// TIA Portal V20 export
// export: Created 2025-12-01T14:56:59.3447129Z, ExportSetting None, DisplayName Totally Integrated Automation Portal, DisplayVersion V20 Update 3, DisplayName TIA Portal Openness, DisplayVersion V20 Update 3, DisplayName TIA Portal Version Control Interface, DisplayVersion V20 Update 3, DisplayName STEP 7 Professional, DisplayVersion V20 Update 3, DisplayName STEP 7 Safety, DisplayVersion V20 Update 2, DisplayName WinCC Basic/Comfort/Advanced, DisplayVersion V20 Update 3, DisplayName WinCC Professional, DisplayVersion V20 Update 3, DisplayName WinCC Unified, DisplayVersion V20 Update 3
FUNCTION "FC402_Conector_ZONA_HB" : Void   // FC402, LAD
{ S7_Optimized_Access := 'FALSE' }
AUTHOR : TLigero
NAME : 20160208
VERSION : 3.1
// stored: AutoNumber false, SetENOAutomatically false
   VAR_INPUT
      Mesa : UInt;
      En_Tension : Bool;
      HB_B_INI : Bool;
      HB_Avance_INI : Bool;
      HB_B_FIN : Bool;
      HB_Avance_FIN : Bool;
      Zona_HB_OK : Bool;
      PRV_AVTF : Bool;
      NXT_Carga_OK : Bool;
      NXT_Avance : Bool;
      V_Paro_Tms : UDInt;
      V_Seg_HB_Avance_Tms : UDInt;
      V_CNTSeparacion : UDInt;
   END_VAR
   VAR_OUTPUT
      PRV_Carga_OK : Bool;
      NXT_AVTF : Bool;
   END_VAR
   VAR_IN_OUT
      Mem_CNT_Tmp_Paro_Tx : Bool;
      Mem_CNT_Seg_HB_Avance : Bool;
      Maux_FN : Bool;
      MemAuxFN_HBpHs : Bool;
   END_VAR
   VAR_TEMP
      OK_Separacion_salida : Bool;
      FN_HBpHs : Bool;
      OK_sep_entrada : Bool;
      TEMP_HB_PTF_Desc : Bool;
      Ok_Tension : Bool;
      EstadoVI : "EstadosMesa";   // Estado del Vehiculo Inteliguente de la Mesa
   END_VAR
   VAR_TEMP   // added for the SCL form of the ladder/FBD networks
      _w1 : Bool;
   END_VAR
BEGIN

REGION Network 1
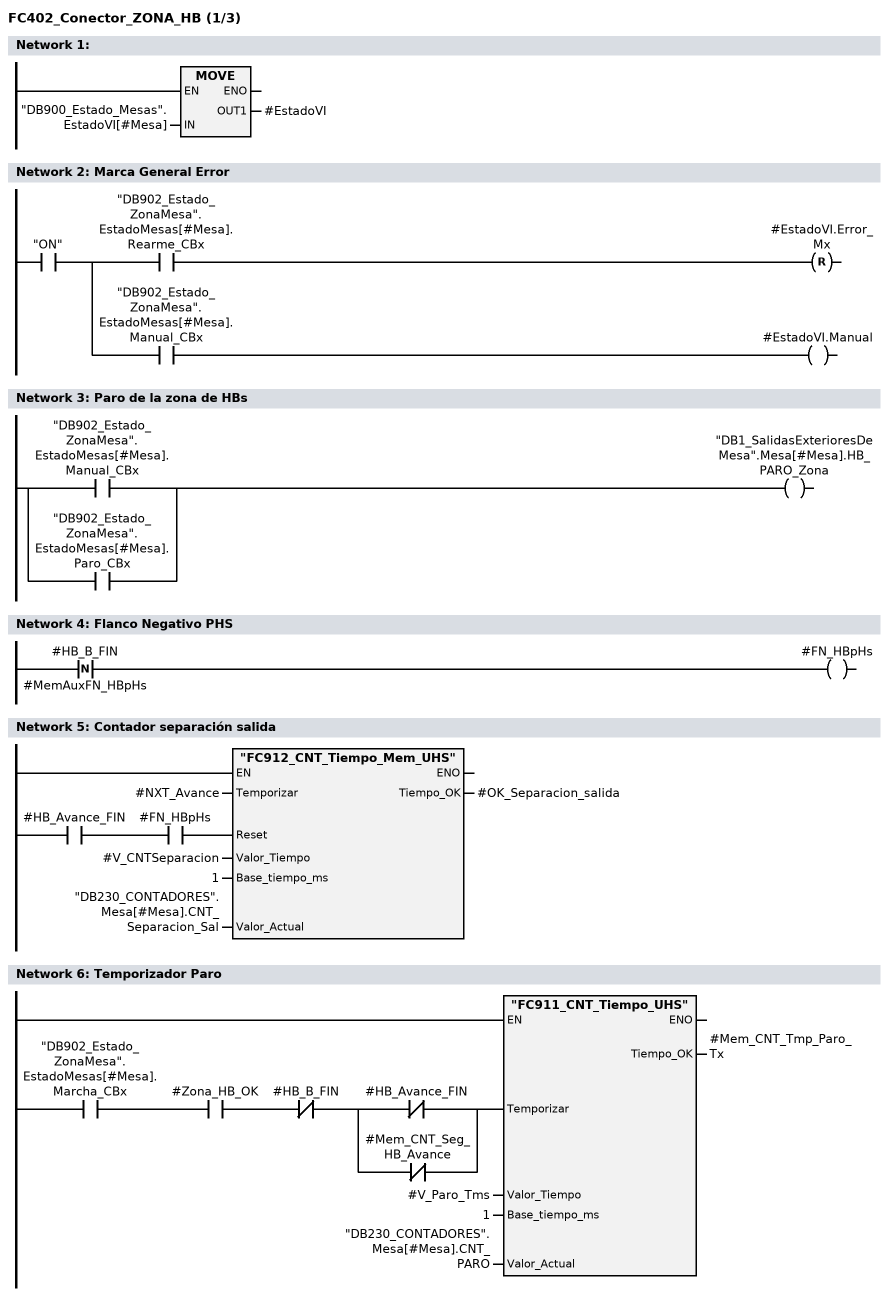
   RUNG wire#powerrail
      Move(in := "DB900_Estado_Mesas".EstadoVI[#Mesa], out1 => #EstadoVI)
   END_RUNG
   // the same network as SCL:
   #EstadoVI := "DB900_Estado_Mesas".EstadoVI[#Mesa];
END_REGION

REGION Network 2: Marca General Error
   RUNG wire#powerrail
      Contact( "ON" )
      wire#w1
      Contact( "DB902_Estado_ZonaMesa".EstadoMesas[#Mesa].Rearme_CBx )
      R_Coil( #EstadoVI.Error_Mx )
   END_RUNG
   RUNG wire#w1
      Contact( "DB902_Estado_ZonaMesa".EstadoMesas[#Mesa].Manual_CBx )
      Coil( #EstadoVI.Manual )
   END_RUNG
   // the same network as SCL:
   IF "ON" AND "DB902_Estado_ZonaMesa".EstadoMesas[#Mesa].Rearme_CBx THEN
       #EstadoVI.Error_Mx := FALSE;
   END_IF;
   #EstadoVI.Manual := "ON" AND "DB902_Estado_ZonaMesa".EstadoMesas[#Mesa].Manual_CBx;
END_REGION

REGION Network 3: Paro de la zona de HBs
   RUNG wire#powerrail
      Contact( "DB902_Estado_ZonaMesa".EstadoMesas[#Mesa].Manual_CBx )
      wire#w1
      Coil( "DB1_SalidasExterioresDeMesa".Mesa[#Mesa].HB_PARO_Zona )
   END_RUNG
   RUNG wire#powerrail
      Contact( "DB902_Estado_ZonaMesa".EstadoMesas[#Mesa].Paro_CBx )
   END_RUNG wire#w1
   // the same network as SCL:
   "DB1_SalidasExterioresDeMesa".Mesa[#Mesa].HB_PARO_Zona := "DB902_Estado_ZonaMesa".EstadoMesas[#Mesa].Manual_CBx OR "DB902_Estado_ZonaMesa".EstadoMesas[#Mesa].Paro_CBx;
END_REGION

REGION Network 4: Flanco Negativo PHS
   RUNG wire#powerrail
      N_Contact(operand := #HB_B_FIN, bit := #MemAuxFN_HBpHs)
      Coil( #FN_HBpHs )
   END_RUNG
   // the same network as SCL:
   #_w1 := NOT #HB_B_FIN AND #MemAuxFN_HBpHs;   // falling edge of #HB_B_FIN
   #MemAuxFN_HBpHs := #HB_B_FIN;
   #FN_HBpHs := #_w1;
END_REGION

REGION Network 5: Contador separación salida
   RUNG wire#powerrail
      "FC912_CNT_Tiempo_Mem_UHS"(Reset := wire#w1, Temporizar := #NXT_Avance, Valor_Tiempo := #V_CNTSeparacion, Base_tiempo_ms := 1, Valor_Actual := "DB230_CONTADORES".Mesa[#Mesa].CNT_Separacion_Sal, Tiempo_OK => #OK_Separacion_salida)
   END_RUNG
   RUNG wire#powerrail
      Contact( #HB_Avance_FIN )
      Contact( #FN_HBpHs )
   END_RUNG wire#w1
   // the same network as SCL:
   "FC912_CNT_Tiempo_Mem_UHS"(Temporizar := #NXT_Avance,
                           Reset := #HB_Avance_FIN AND #FN_HBpHs,
                           Valor_Tiempo := #V_CNTSeparacion,
                           Base_tiempo_ms := 1,
                           Valor_Actual := "DB230_CONTADORES".Mesa[#Mesa].CNT_Separacion_Sal,
                           Tiempo_OK => #OK_Separacion_salida);
END_REGION

REGION Network 6: Temporizador Paro
   RUNG wire#powerrail
      "FC911_CNT_Tiempo_UHS"(Temporizar := wire#w2, Valor_Tiempo := #V_Paro_Tms, Base_tiempo_ms := 1, Valor_Actual := "DB230_CONTADORES".Mesa[#Mesa].CNT_PARO, Tiempo_OK => #Mem_CNT_Tmp_Paro_Tx)
   END_RUNG
   RUNG wire#powerrail
      Contact( "DB902_Estado_ZonaMesa".EstadoMesas[#Mesa].Marcha_CBx )
      Contact( #Zona_HB_OK )
      I_Contact( #HB_B_FIN )
      wire#w1
      I_Contact( #HB_Avance_FIN )
   END_RUNG wire#w2
   RUNG wire#w1
      I_Contact( #Mem_CNT_Seg_HB_Avance )
   END_RUNG wire#w2
   // the same network as SCL:
   "FC911_CNT_Tiempo_UHS"(Temporizar := "DB902_Estado_ZonaMesa".EstadoMesas[#Mesa].Marcha_CBx AND #Zona_HB_OK AND NOT #HB_B_FIN AND (NOT #HB_Avance_FIN OR NOT #Mem_CNT_Seg_HB_Avance),
                          Valor_Tiempo := #V_Paro_Tms,
                          Base_tiempo_ms := 1,
                          Valor_Actual := "DB230_CONTADORES".Mesa[#Mesa].CNT_PARO,
                          Tiempo_OK => #Mem_CNT_Tmp_Paro_Tx);
END_REGION

REGION Network 7: Permiso descarga
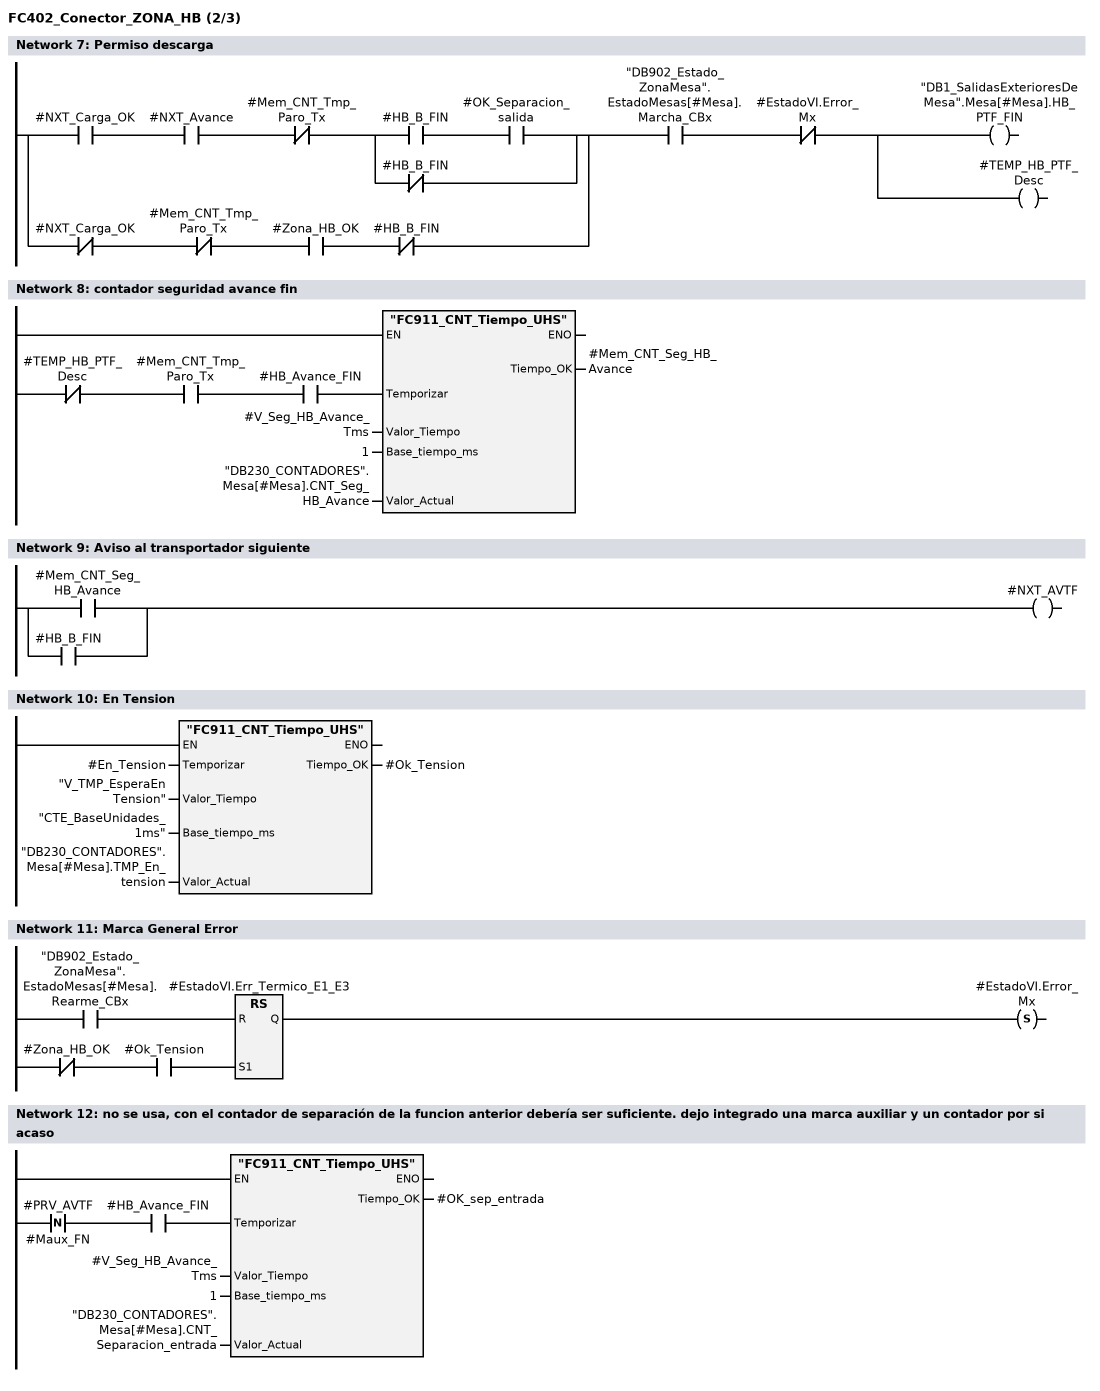
   RUNG wire#powerrail
      Contact( #NXT_Carga_OK )
      Contact( #NXT_Avance )
      I_Contact( #Mem_CNT_Tmp_Paro_Tx )
      wire#w1
      Contact( #HB_B_FIN )
      Contact( #OK_Separacion_salida )
      wire#w2
      Contact( "DB902_Estado_ZonaMesa".EstadoMesas[#Mesa].Marcha_CBx )
      I_Contact( #EstadoVI.Error_Mx )
      wire#w3
      Coil( "DB1_SalidasExterioresDeMesa".Mesa[#Mesa].HB_PTF_FIN )
   END_RUNG
   RUNG wire#w1
      I_Contact( #HB_B_FIN )
   END_RUNG wire#w2
   RUNG wire#powerrail
      I_Contact( #NXT_Carga_OK )
      I_Contact( #Mem_CNT_Tmp_Paro_Tx )
      Contact( #Zona_HB_OK )
      I_Contact( #HB_B_FIN )
   END_RUNG wire#w2
   RUNG wire#w3
      Coil( #TEMP_HB_PTF_Desc )
   END_RUNG
   // the same network as SCL:
   #_w1 := ((#NXT_Carga_OK AND #NXT_Avance AND NOT #Mem_CNT_Tmp_Paro_Tx AND ((#HB_B_FIN AND #OK_Separacion_salida) OR NOT #HB_B_FIN)) OR (NOT #NXT_Carga_OK AND NOT #Mem_CNT_Tmp_Paro_Tx AND #Zona_HB_OK AND NOT #HB_B_FIN)) AND "DB902_Estado_ZonaMesa".EstadoMesas[#Mesa].Marcha_CBx AND NOT #EstadoVI.Error_Mx;
   "DB1_SalidasExterioresDeMesa".Mesa[#Mesa].HB_PTF_FIN := ((#NXT_Carga_OK AND #NXT_Avance AND NOT #Mem_CNT_Tmp_Paro_Tx AND ((#HB_B_FIN AND #OK_Separacion_salida) OR NOT #HB_B_FIN)) OR (NOT #NXT_Carga_OK AND NOT #Mem_CNT_Tmp_Paro_Tx AND #Zona_HB_OK AND NOT #HB_B_FIN)) AND "DB902_Estado_ZonaMesa".EstadoMesas[#Mesa].Marcha_CBx AND NOT #EstadoVI.Error_Mx;
   #TEMP_HB_PTF_Desc := #_w1;
END_REGION

REGION Network 8: contador seguridad avance fin
   RUNG wire#powerrail
      "FC911_CNT_Tiempo_UHS"(Temporizar := wire#w1, Valor_Tiempo := #V_Seg_HB_Avance_Tms, Base_tiempo_ms := 1, Valor_Actual := "DB230_CONTADORES".Mesa[#Mesa].CNT_Seg_HB_Avance, Tiempo_OK => #Mem_CNT_Seg_HB_Avance)
   END_RUNG
   RUNG wire#powerrail
      I_Contact( #TEMP_HB_PTF_Desc )
      Contact( #Mem_CNT_Tmp_Paro_Tx )
      Contact( #HB_Avance_FIN )
   END_RUNG wire#w1
   // the same network as SCL:
   "FC911_CNT_Tiempo_UHS"(Temporizar := NOT #TEMP_HB_PTF_Desc AND #Mem_CNT_Tmp_Paro_Tx AND #HB_Avance_FIN,
                          Valor_Tiempo := #V_Seg_HB_Avance_Tms,
                          Base_tiempo_ms := 1,
                          Valor_Actual := "DB230_CONTADORES".Mesa[#Mesa].CNT_Seg_HB_Avance,
                          Tiempo_OK => #Mem_CNT_Seg_HB_Avance);
END_REGION

REGION Network 9: Aviso al transportador siguiente
   RUNG wire#powerrail
      Contact( #Mem_CNT_Seg_HB_Avance )
      wire#w1
      Coil( #NXT_AVTF )
   END_RUNG
   RUNG wire#powerrail
      Contact( #HB_B_FIN )
   END_RUNG wire#w1
   // the same network as SCL:
   #NXT_AVTF := #Mem_CNT_Seg_HB_Avance OR #HB_B_FIN;
END_REGION

REGION Network 10: En Tension
   RUNG wire#powerrail
      "FC911_CNT_Tiempo_UHS"(Temporizar := #En_Tension, Valor_Tiempo := "V_TMP_EsperaEnTension", Base_tiempo_ms := "CTE_BaseUnidades_1ms", Valor_Actual := "DB230_CONTADORES".Mesa[#Mesa].TMP_En_tension, Tiempo_OK => #Ok_Tension)
   END_RUNG
   // the same network as SCL:
   "FC911_CNT_Tiempo_UHS"(Temporizar := #En_Tension,
                          Valor_Tiempo := "V_TMP_EsperaEnTension",
                          Base_tiempo_ms := "CTE_BaseUnidades_1ms",
                          Valor_Actual := "DB230_CONTADORES".Mesa[#Mesa].TMP_En_tension,
                          Tiempo_OK => #Ok_Tension);
END_REGION

REGION Network 11: Marca General Error
   RUNG wire#powerrail
      Contact( "DB902_Estado_ZonaMesa".EstadoMesas[#Mesa].Rearme_CBx )
      S_RS(operand := #EstadoVI.Err_Termico_E1_E3, s1 := wire#w1)
      S_Coil( #EstadoVI.Error_Mx )
   END_RUNG
   RUNG wire#powerrail
      I_Contact( #Zona_HB_OK )
      Contact( #Ok_Tension )
   END_RUNG wire#w1
   // the same network as SCL:
   IF "DB902_Estado_ZonaMesa".EstadoMesas[#Mesa].Rearme_CBx THEN
       #EstadoVI.Err_Termico_E1_E3 := FALSE;   // RS flip-flop
   END_IF;
   IF NOT #Zona_HB_OK AND #Ok_Tension THEN #EstadoVI.Err_Termico_E1_E3 := TRUE; END_IF;
   IF #EstadoVI.Err_Termico_E1_E3 THEN #EstadoVI.Error_Mx := TRUE; END_IF;
END_REGION

REGION Network 12: no se usa, con el contador de separación de la funcion anterior debería ser suficiente. dejo integrado una marca auxiliar y un contador por si acaso
   RUNG wire#powerrail
      "FC911_CNT_Tiempo_UHS"(Temporizar := wire#w1, Valor_Tiempo := #V_Seg_HB_Avance_Tms, Base_tiempo_ms := 1, Valor_Actual := "DB230_CONTADORES".Mesa[#Mesa].CNT_Separacion_entrada, Tiempo_OK => #OK_sep_entrada)
   END_RUNG
   RUNG wire#powerrail
      N_Contact(operand := #PRV_AVTF, bit := #Maux_FN)
      Contact( #HB_Avance_FIN )
   END_RUNG wire#w1
   // the same network as SCL:
   #_w1 := NOT #PRV_AVTF AND #Maux_FN;   // falling edge of #PRV_AVTF
   #Maux_FN := #PRV_AVTF;
   "FC911_CNT_Tiempo_UHS"(Temporizar := #_w1 AND #HB_Avance_FIN,
                          Valor_Tiempo := #V_Seg_HB_Avance_Tms,
                          Base_tiempo_ms := 1,
                          Valor_Actual := "DB230_CONTADORES".Mesa[#Mesa].CNT_Separacion_entrada,
                          Tiempo_OK => #OK_sep_entrada);
END_REGION

REGION Network 13: interlock transportador inicial
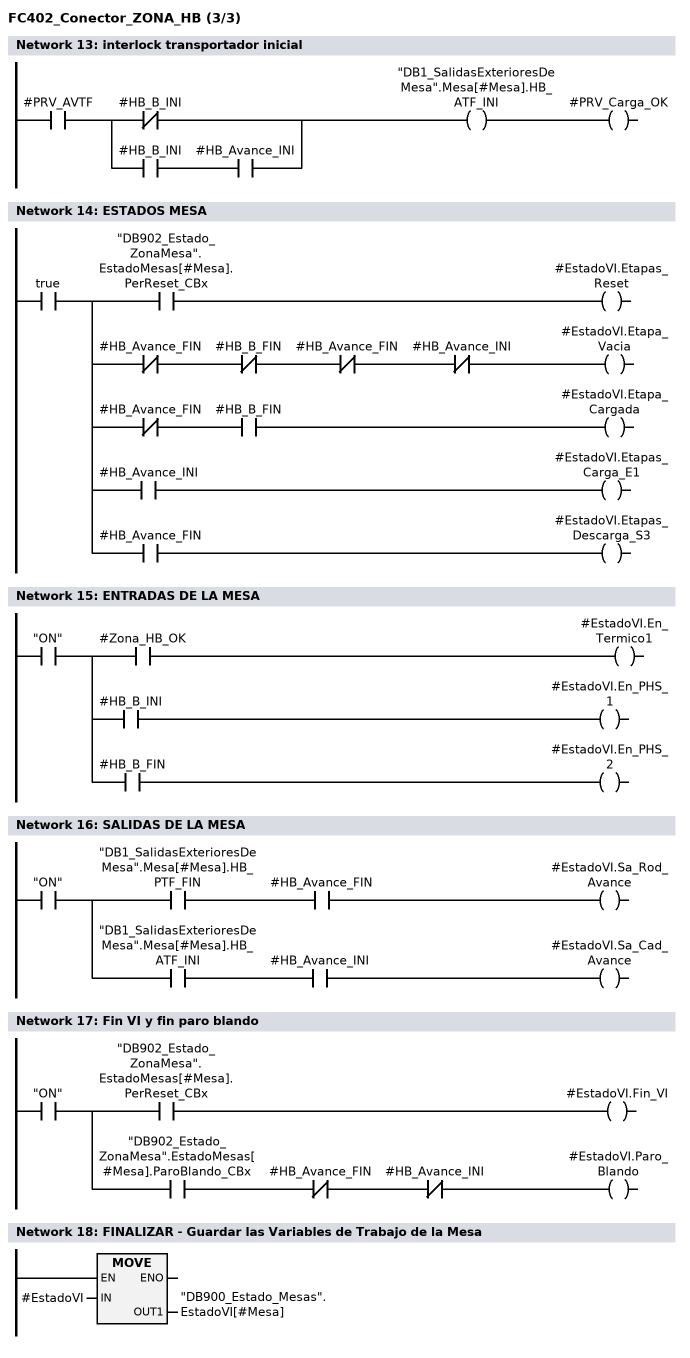
   RUNG wire#powerrail
      Contact( #PRV_AVTF )
      wire#w1
      I_Contact( #HB_B_INI )
      wire#w2
      Coil( "DB1_SalidasExterioresDeMesa".Mesa[#Mesa].HB_ATF_INI )
      Coil( #PRV_Carga_OK )
   END_RUNG
   RUNG wire#w1
      Contact( #HB_B_INI )
      Contact( #HB_Avance_INI )
   END_RUNG wire#w2
   // the same network as SCL:
   "DB1_SalidasExterioresDeMesa".Mesa[#Mesa].HB_ATF_INI := #PRV_AVTF AND (NOT #HB_B_INI OR (#HB_B_INI AND #HB_Avance_INI));
   #PRV_Carga_OK := #PRV_AVTF AND (NOT #HB_B_INI OR (#HB_B_INI AND #HB_Avance_INI));
END_REGION

REGION Network 14: ESTADOS MESA
   RUNG wire#powerrail
      Contact( true )
      wire#w1
      Contact( "DB902_Estado_ZonaMesa".EstadoMesas[#Mesa].PerReset_CBx )
      Coil( #EstadoVI.Etapas_Reset )
   END_RUNG
   RUNG wire#w1
      I_Contact( #HB_Avance_FIN )
      I_Contact( #HB_B_FIN )
      I_Contact( #HB_Avance_FIN )
      I_Contact( #HB_Avance_INI )
      Coil( #EstadoVI.Etapa_Vacia )
   END_RUNG
   RUNG wire#w1
      I_Contact( #HB_Avance_FIN )
      Contact( #HB_B_FIN )
      Coil( #EstadoVI.Etapa_Cargada )
   END_RUNG
   RUNG wire#w1
      Contact( #HB_Avance_INI )
      Coil( #EstadoVI.Etapas_Carga_E1 )
   END_RUNG
   RUNG wire#w1
      Contact( #HB_Avance_FIN )
      Coil( #EstadoVI.Etapas_Descarga_S3 )
   END_RUNG
   // the same network as SCL:
   #EstadoVI.Etapas_Reset := true AND "DB902_Estado_ZonaMesa".EstadoMesas[#Mesa].PerReset_CBx;
   #EstadoVI.Etapa_Vacia := true AND NOT #HB_Avance_FIN AND NOT #HB_B_FIN AND NOT #HB_Avance_FIN AND NOT #HB_Avance_INI;
   #EstadoVI.Etapa_Cargada := true AND NOT #HB_Avance_FIN AND #HB_B_FIN;
   #EstadoVI.Etapas_Carga_E1 := true AND #HB_Avance_INI;
   #EstadoVI.Etapas_Descarga_S3 := true AND #HB_Avance_FIN;
END_REGION

REGION Network 15: ENTRADAS DE LA MESA
   RUNG wire#powerrail
      Contact( "ON" )
      wire#w1
      Contact( #Zona_HB_OK )
      Coil( #EstadoVI.En_Termico1 )
   END_RUNG
   RUNG wire#w1
      Contact( #HB_B_INI )
      Coil( #EstadoVI.En_PHS_1 )
   END_RUNG
   RUNG wire#w1
      Contact( #HB_B_FIN )
      Coil( #EstadoVI.En_PHS_2 )
   END_RUNG
   // the same network as SCL:
   #EstadoVI.En_Termico1 := "ON" AND #Zona_HB_OK;
   #EstadoVI.En_PHS_1 := "ON" AND #HB_B_INI;
   #EstadoVI.En_PHS_2 := "ON" AND #HB_B_FIN;
END_REGION

REGION Network 16: SALIDAS DE LA MESA
   RUNG wire#powerrail
      Contact( "ON" )
      wire#w1
      Contact( "DB1_SalidasExterioresDeMesa".Mesa[#Mesa].HB_PTF_FIN )
      Contact( #HB_Avance_FIN )
      Coil( #EstadoVI.Sa_Rod_Avance )
   END_RUNG
   RUNG wire#w1
      Contact( "DB1_SalidasExterioresDeMesa".Mesa[#Mesa].HB_ATF_INI )
      Contact( #HB_Avance_INI )
      Coil( #EstadoVI.Sa_Cad_Avance )
   END_RUNG
   // the same network as SCL:
   #EstadoVI.Sa_Rod_Avance := "ON" AND "DB1_SalidasExterioresDeMesa".Mesa[#Mesa].HB_PTF_FIN AND #HB_Avance_FIN;
   #EstadoVI.Sa_Cad_Avance := "ON" AND "DB1_SalidasExterioresDeMesa".Mesa[#Mesa].HB_ATF_INI AND #HB_Avance_INI;
END_REGION

REGION Network 17: Fin VI y fin paro blando
   RUNG wire#powerrail
      Contact( "ON" )
      wire#w1
      Contact( "DB902_Estado_ZonaMesa".EstadoMesas[#Mesa].PerReset_CBx )
      Coil( #EstadoVI.Fin_VI )
   END_RUNG
   RUNG wire#w1
      Contact( "DB902_Estado_ZonaMesa".EstadoMesas[#Mesa].ParoBlando_CBx )
      I_Contact( #HB_Avance_FIN )
      I_Contact( #HB_Avance_INI )
      Coil( #EstadoVI.Paro_Blando )
   END_RUNG
   // the same network as SCL:
   #EstadoVI.Fin_VI := "ON" AND "DB902_Estado_ZonaMesa".EstadoMesas[#Mesa].PerReset_CBx;
   #EstadoVI.Paro_Blando := "ON" AND "DB902_Estado_ZonaMesa".EstadoMesas[#Mesa].ParoBlando_CBx AND NOT #HB_Avance_FIN AND NOT #HB_Avance_INI;
END_REGION

REGION Network 18: FINALIZAR - Guardar las Variables de Trabajo de la Mesa
   RUNG wire#powerrail
      Move(in := #EstadoVI, out1 => "DB900_Estado_Mesas".EstadoVI[#Mesa])
   END_RUNG
   // the same network as SCL:
   "DB900_Estado_Mesas".EstadoVI[#Mesa] := #EstadoVI;
END_REGION
END_FUNCTION
